FUNCTION_BLOCK OutputCompressor (* Basic Function Block Type *)
  (* Standard: 61499-2 *)
  (* Version 0.0, 11/2/2016, Dmitry, nxtControl GmbH, Template *)
  PACKAGE Main;
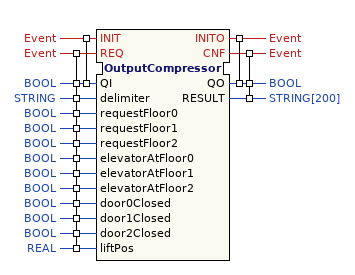
  EVENT_INPUT
    INIT WITH QI; (* Initialization Request *)
    REQ WITH QI, delimiter, requestFloor0, requestFloor1, requestFloor2, elevatorAtFloor0, elevatorAtFloor1, elevatorAtFloor2, door0Closed, door1Closed, door2Closed, liftPos; (* Normal Execution Request *)
  END_EVENT
  EVENT_OUTPUT
    INITO WITH QO; (* Initialization Confirm *)
    CNF WITH QO, RESULT; (* Execution Confirmation *)
  END_EVENT
  VAR_INPUT
    QI : BOOL; (* Input event qualifier *)
    delimiter : STRING;
    requestFloor0 : BOOL;
    requestFloor1 : BOOL;
    requestFloor2 : BOOL;
    elevatorAtFloor0 : BOOL;
    elevatorAtFloor1 : BOOL;
    elevatorAtFloor2 : BOOL;
    door0Closed : BOOL;
    door1Closed : BOOL;
    door2Closed : BOOL;
    liftPos : REAL;
  END_VAR
  VAR_OUTPUT
    QO : BOOL; (* Output event qualifier *)
    RESULT : STRING[200];
  END_VAR
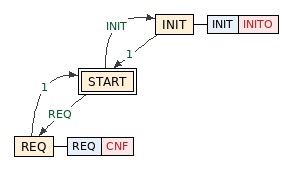
  EC_STATES
    START; (* Initial State *)
    INIT : INIT -> INITO; (* Initialization *)
    REQ : REQ -> CNF; (* Normal execution *)
  END_STATES
  EC_TRANSITIONS
    START TO INIT := INIT;
    INIT TO START := 1;
    START TO REQ := REQ;
    REQ TO START := 1;
  END_TRANSITIONS
  ALGORITHM INIT IN ST: (* Initialization algorithm *)
QO := TRUE;
  END_ALGORITHM
  ALGORITHM REQ IN ST: (* Normally executed algorithm *)
RESULT :=
CONCAT(
  (*CONCAT(
    BOOL_TO_STRING(buttonFloor0), delimiter,
    BOOL_TO_STRING(buttonFloor1), delimiter,
    BOOL_TO_STRING(buttonFloor2), delimiter
  ),*)
  CONCAT(
    BOOL_TO_STRING(requestFloor0), delimiter,
    BOOL_TO_STRING(requestFloor1), delimiter,
    BOOL_TO_STRING(requestFloor2), delimiter
  ),
  CONCAT(
    BOOL_TO_STRING(elevatorAtFloor0), delimiter,
    BOOL_TO_STRING(elevatorAtFloor1), delimiter,
    BOOL_TO_STRING(elevatorAtFloor2), delimiter
  ),
  CONCAT(
    BOOL_TO_STRING(door0Closed), delimiter,
    BOOL_TO_STRING(door1Closed), delimiter,
    BOOL_TO_STRING(door2Closed), delimiter
  ),
  CONCAT(
    REAL_TO_STRING(liftPos), delimiter
  ),
  "$N"
);
  END_ALGORITHM
END_FUNCTION_BLOCK
